(* IEC 61131-3 sources: CodesysTest/export/Function Blocks/FB_Fault/FB_Fault.pou/InstanceName.prop, 1 file *)

(* ---- Set.pm.st ---- *)
(*#-#-#-#-#-#-#-#-#-#---Declaration---#-#-#-#-#-#-#-#-#-#-#-#-#*)

VAR
END_VAR
(*#-#-#-#-#-#-#-#-#-#---Implementation---#-#-#-#-#-#-#-#-#-#-#-#-#*)

_instanceName := InstanceName;
